// TIA Portal V15.1 export
// export: Created 2026-01-09T13:45:13.784524Z, ExportSetting WithDefaults, WithReadOnly, DisplayName Totally Integrated Automation Portal, DisplayVersion V15.1 Update 8, DisplayName TIA Portal Openness, DisplayVersion V15.1 Update 8, DisplayName STEP 7 Professional, DisplayVersion V15.1 Update 8, DisplayName WinCC Advanced, DisplayVersion V15.1 Update 8
DATA_BLOCK "10.1.RUNG_CE1"   // DB1006
{ S7_Optimized_Access := 'TRUE' }
VERSION : 0.1
// stored: AutoNumber false, CodeModifiedDate 2025-08-27T17:14:35.1936779Z, CompileDate 2025-08-30T17:40:35.2998011Z, CreationDate 2024-10-12T12:36:08.0193576Z, DBAccessibleFromOPCUA true, DownloadWithoutReinit false, InstanceOfName 10.TIMER_CLOCK, InstanceOfNumber 10, InstanceOfType FB, InterfaceModifiedDate 2023-08-14T08:08:19.3737097Z, IsConsistent true, IsKnowHowProtected false, IsRetainMemResEnabled false, MemoryReserve 100, ModifiedDate 2025-08-27T17:14:35.1936779Z, ParameterModified 2022-05-24T16:04:05.0982286Z, StructureModified 2023-08-14T08:08:19.3737097Z, UDAEnableTagReadback false
"10.TIMER_CLOCK"
   // VAR_INPUT
   //    ON : Bool;
   //    CLOCK_1S : Bool;
   //    T_ON : Real;
   //    T_OFF : Real;
   // END_VAR
   // VAR_OUTPUT
   //    OUT : Bool;
   // END_VAR
   // VAR RETAIN
   //    TON : Real;
   //    TOFF : Real;
   // END_VAR
   // VAR
   //    CLK1 : Bool;
   // END_VAR
BEGIN
END_DATA_BLOCK
